FUNCTION_BLOCK MPC_MOVE_BLOCKED_NMPC_V4 (* High-range V4 state-disturbance MPC identified from real 3, 5, 8.5 and 13 cm calibration transients *)
  (* Standard: 61499-2 *)
  (* Version 4.0, 2026-08-29, Guilherme *)
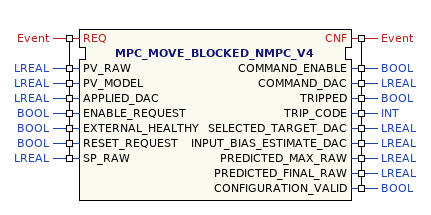
  EVENT_INPUT
    REQ WITH PV_RAW, PV_MODEL, APPLIED_DAC, ENABLE_REQUEST, EXTERNAL_HEALTHY, RESET_REQUEST, SP_RAW; (* Execute one 500 ms high-range MPC V4 cycle *)
  END_EVENT
  EVENT_OUTPUT
    CNF WITH COMMAND_ENABLE, COMMAND_DAC, TRIPPED, TRIP_CODE, SELECTED_TARGET_DAC, INPUT_BIAS_ESTIMATE_DAC, PREDICTED_MAX_RAW, PREDICTED_FINAL_RAW, CONFIGURATION_VALID; (* MPC cycle completed *)
  END_EVENT
  VAR_INPUT
    PV_RAW : LREAL; (* Unfiltered raw level used by the measured hard trip *)
    PV_MODEL : LREAL; (* 9-sample rolling-median raw level used by the identified model *)
    APPLIED_DAC : LREAL; (* PLC-confirmed DAC used as the move-constraint reference *)
    ENABLE_REQUEST : BOOL; (* Explicit operator/commissioning enable; FALSE is normal zero-output mode *)
    EXTERNAL_HEALTHY : BOOL; (* PLC/gateway watchdog healthy input *)
    RESET_REQUEST : BOOL; (* Explicitly clear the latched MPC trip and internal estimator state *)
    SP_RAW : LREAL; (* Raw-count setpoint; 15 cm validation target is 16000 *)
  END_VAR
  VAR_OUTPUT
    COMMAND_ENABLE : BOOL; (* Fail-closed actuator enable request *)
    COMMAND_DAC : LREAL; (* MPC DAC request before downstream defense-in-depth limiting *)
    TRIPPED : BOOL; (* Latched MPC trip state *)
    TRIP_CODE : INT; (* 0=none,1=non-finite input,2=external health,3=PV bounds,4=AppliedDAC bounds,5=setpoint bounds,6=no feasible prediction,7=delay history not ready *)
    SELECTED_TARGET_DAC : LREAL; (* Move-blocked target selected by the current horizon search *)
    INPUT_BIAS_ESTIMATE_DAC : LREAL; (* Bounded offset-compensation estimate *)
    PREDICTED_MAX_RAW : LREAL; (* Maximum predicted model level for the selected candidate *)
    PREDICTED_FINAL_RAW : LREAL; (* Final horizon model level for the selected candidate *)
    CONFIGURATION_VALID : BOOL; (* Frozen V4 high-range configuration is internally valid *)
  END_VAR
  VAR
    trip_latched_internal : BOOL := FALSE;
    trip_code_internal : INT := 0;
    history_count : DINT := 0;
    record_history_internal : BOOL := FALSE;
    best_found : BOOL := FALSE;
    candidate_feasible : BOOL := FALSE;
    h00 : LREAL := 0.0;
    h01 : LREAL := 0.0;
    h02 : LREAL := 0.0;
    h03 : LREAL := 0.0;
    h04 : LREAL := 0.0;
    h05 : LREAL := 0.0;
    h06 : LREAL := 0.0;
    h07 : LREAL := 0.0;
    h08 : LREAL := 0.0;
    h09 : LREAL := 0.0;
    h10 : LREAL := 0.0;
    h11 : LREAL := 0.0;
    h12 : LREAL := 0.0;
    h13 : LREAL := 0.0;
    h14 : LREAL := 0.0;
    h15 : LREAL := 0.0;
    h16 : LREAL := 0.0;
    h17 : LREAL := 0.0;
    q00 : LREAL := 0.0;
    q01 : LREAL := 0.0;
    q02 : LREAL := 0.0;
    q03 : LREAL := 0.0;
    q04 : LREAL := 0.0;
    q05 : LREAL := 0.0;
    q06 : LREAL := 0.0;
    q07 : LREAL := 0.0;
    q08 : LREAL := 0.0;
    q09 : LREAL := 0.0;
    q10 : LREAL := 0.0;
    q11 : LREAL := 0.0;
    q12 : LREAL := 0.0;
    q13 : LREAL := 0.0;
    q14 : LREAL := 0.0;
    q15 : LREAL := 0.0;
    q16 : LREAL := 0.0;
    q17 : LREAL := 0.0;
    best_cost : LREAL := 0.0;
    best_target : LREAL := 0.0;
    best_predicted_max : LREAL := 0.0;
    best_predicted_final : LREAL := 0.0;
    candidate_target : LREAL := 0.0;
    predicted_y : LREAL := 0.0;
    predicted_u : LREAL := 0.0;
    previous_u : LREAL := 0.0;
    delayed_u : LREAL := 0.0;
    candidate_cost : LREAL := 0.0;
    candidate_predicted_max : LREAL := 0.0;
    delta_u : LREAL := 0.0;
    effective_input : LREAL := 0.0;
    phi_value : LREAL := 0.0;
    tracking_error : LREAL := 0.0;
    move_value : LREAL := 0.0;
    soft_excess : LREAL := 0.0;
    terminal_error : LREAL := 0.0;
    command_candidate : LREAL := 0.0;
    candidate_index : DINT := 0;
    prediction_index : DINT := 0;
    disturbance_hat_internal : LREAL := 0.0;
    disturbance_previous_pv_internal : LREAL := 0.0;
    disturbance_previous_valid_internal : BOOL := FALSE;
    disturbance_prediction_internal : LREAL := 0.0;
    disturbance_innovation_internal : LREAL := 0.0;
  END_VAR
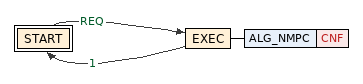
  EC_STATES
    START;
    EXEC : ALG_NMPC -> CNF;
  END_STATES
  EC_TRANSITIONS
    START TO EXEC := REQ;
    EXEC TO START := 1;
  END_TRANSITIONS
  ALGORITHM ALG_NMPC IN ST: (* Move-blocked V4 high-range NMPC with state-disturbance estimation, model constraints, trip latch, and piecewise-linear x^1.2 input *)
IF RESET_REQUEST THEN
    trip_latched_internal := FALSE;
    trip_code_internal := 0;
    disturbance_hat_internal := LREAL#0.0;
    disturbance_previous_pv_internal := LREAL#0.0;
    disturbance_previous_valid_internal := FALSE;
    disturbance_prediction_internal := LREAL#0.0;
    disturbance_innovation_internal := LREAL#0.0;
END_IF;

CONFIGURATION_VALID := TRUE;
COMMAND_ENABLE := FALSE;
COMMAND_DAC := LREAL#0.0;
SELECTED_TARGET_DAC := LREAL#0.0;
INPUT_BIAS_ESTIMATE_DAC := LREAL#0.0;
PREDICTED_MAX_RAW := LREAL#-1.0;
PREDICTED_FINAL_RAW := LREAL#-1.0;

record_history_internal := (PV_RAW = PV_RAW) AND (PV_MODEL = PV_MODEL) AND (APPLIED_DAC = APPLIED_DAC) AND (SP_RAW = SP_RAW) AND (APPLIED_DAC >= LREAL#0.0) AND (APPLIED_DAC <= LREAL#16000.0);

IF NOT trip_latched_internal THEN
    IF NOT ENABLE_REQUEST THEN
        disturbance_hat_internal := LREAL#0.0;
        disturbance_previous_pv_internal := LREAL#0.0;
        disturbance_previous_valid_internal := FALSE;
        disturbance_prediction_internal := LREAL#0.0;
        disturbance_innovation_internal := LREAL#0.0;
        COMMAND_ENABLE := FALSE;
        COMMAND_DAC := LREAL#0.0;
    ELSE
        IF NOT EXTERNAL_HEALTHY THEN
            trip_latched_internal := TRUE;
            trip_code_internal := 2;
        ELSIF NOT (PV_RAW = PV_RAW) OR NOT (PV_MODEL = PV_MODEL) OR NOT (APPLIED_DAC = APPLIED_DAC) OR NOT (SP_RAW = SP_RAW) THEN
            trip_latched_internal := TRUE;
            trip_code_internal := 1;
        ELSIF PV_RAW < LREAL#0.0 OR PV_MODEL < LREAL#0.0 OR PV_RAW >= LREAL#20000.0 THEN
            trip_latched_internal := TRUE;
            trip_code_internal := 3;
        ELSIF APPLIED_DAC < LREAL#0.0 OR APPLIED_DAC > LREAL#16000.0 THEN
            trip_latched_internal := TRUE;
            trip_code_internal := 4;
        ELSIF SP_RAW < LREAL#0.0 OR SP_RAW >= LREAL#18000.0 THEN
            trip_latched_internal := TRUE;
            trip_code_internal := 5;
        ELSE
            IF disturbance_previous_valid_internal THEN
                IF disturbance_previous_pv_internal < LREAL#257.0 THEN
                    disturbance_previous_pv_internal := LREAL#257.0;
                END_IF;
                effective_input := APPLIED_DAC - LREAL#11750.0;
                IF effective_input < LREAL#0.0 THEN
                    effective_input := LREAL#0.0;
                ELSIF effective_input > LREAL#4250.0 THEN
                    effective_input := LREAL#4250.0;
                END_IF;
                IF effective_input <= LREAL#0.0 THEN
                    phi_value := LREAL#0.0;
                ELSIF effective_input <= LREAL#250.0 THEN
                    phi_value := LREAL#0.000000000000000 + LREAL#3.017088168272581 * (effective_input - LREAL#0.0);
                ELSIF effective_input <= LREAL#500.0 THEN
                    phi_value := LREAL#754.272042068145197 + LREAL#3.914360263278881 * (effective_input - LREAL#250.0);
                ELSIF effective_input <= LREAL#750.0 THEN
                    phi_value := LREAL#1732.862107887865477 + LREAL#4.343991804743724 * (effective_input - LREAL#500.0);
                ELSIF effective_input <= LREAL#1000.0 THEN
                    phi_value := LREAL#2818.860059073796492 + LREAL#4.648846585844700 * (effective_input - LREAL#750.0);
                ELSIF effective_input <= LREAL#1250.0 THEN
                    phi_value := LREAL#3981.071705534971443 + LREAL#4.889543362906937 * (effective_input - LREAL#1000.0);
                ELSIF effective_input <= LREAL#1500.0 THEN
                    phi_value := LREAL#5203.457546261705829 + LREAL#5.090329117552494 * (effective_input - LREAL#1250.0);
                ELSIF effective_input <= LREAL#1750.0 THEN
                    phi_value := LREAL#6476.039825649829254 + LREAL#5.263604911708677 * (effective_input - LREAL#1500.0);
                ELSIF effective_input <= LREAL#2000.0 THEN
                    phi_value := LREAL#7791.941053576998456 + LREAL#5.416639939878100 * (effective_input - LREAL#1750.0);
                ELSIF effective_input <= LREAL#2250.0 THEN
                    phi_value := LREAL#9146.101038546523341 + LREAL#5.554090126229741 * (effective_input - LREAL#2000.0);
                ELSIF effective_input <= LREAL#2500.0 THEN
                    phi_value := LREAL#10534.623570103958627 + LREAL#5.679130709085999 * (effective_input - LREAL#2250.0);
                ELSIF effective_input <= LREAL#2750.0 THEN
                    phi_value := LREAL#11954.406247375458406 + LREAL#5.794031214691713 * (effective_input - LREAL#2500.0);
                ELSIF effective_input <= LREAL#3000.0 THEN
                    phi_value := LREAL#13402.914051048386682 + LREAL#5.900474152760405 * (effective_input - LREAL#2750.0);
                ELSIF effective_input <= LREAL#3250.0 THEN
                    phi_value := LREAL#14878.032589238488072 + LREAL#5.999743896709013 * (effective_input - LREAL#3000.0);
                ELSIF effective_input <= LREAL#3500.0 THEN
                    phi_value := LREAL#16377.968563415741301 + LREAL#6.092844710159137 * (effective_input - LREAL#3250.0);
                ELSIF effective_input <= LREAL#3750.0 THEN
                    phi_value := LREAL#17901.179740955525631 + LREAL#6.180577736426479 * (effective_input - LREAL#3500.0);
                ELSIF effective_input <= LREAL#4000.0 THEN
                    phi_value := LREAL#19446.324175062145514 + LREAL#6.263593040671942 * (effective_input - LREAL#3750.0);
                ELSIF effective_input <= LREAL#4250.0 THEN
                    phi_value := LREAL#21012.222435230130941 + LREAL#6.342425861622032 * (effective_input - LREAL#4000.0);
                ELSE
                    phi_value := LREAL#22597.828900635639002;
                END_IF;
                disturbance_prediction_internal := LREAL#257.0 + LREAL#0.997231776304349 * (disturbance_previous_pv_internal - LREAL#257.0) + LREAL#0.004607840412330 * phi_value;
                disturbance_innovation_internal := PV_MODEL - disturbance_prediction_internal;
                disturbance_hat_internal := LREAL#0.9 * disturbance_hat_internal + LREAL#0.1 * disturbance_innovation_internal;
                IF disturbance_hat_internal > LREAL#10.0 THEN
                    disturbance_hat_internal := LREAL#10.0;
                ELSIF disturbance_hat_internal < LREAL#-10.0 THEN
                    disturbance_hat_internal := LREAL#-10.0;
                END_IF;
            END_IF;
            disturbance_previous_pv_internal := PV_MODEL;
            disturbance_previous_valid_internal := TRUE;
            best_found := FALSE;
            best_cost := LREAL#1000000000.0;
            best_target := LREAL#0.0;
            best_predicted_max := LREAL#-1.0;
            best_predicted_final := LREAL#-1.0;
            FOR candidate_index := 0 TO 10 DO
                CASE candidate_index OF
                    0:
                        candidate_target := LREAL#0.0;
                    1:
                        candidate_target := LREAL#12000.0;
                    2:
                        candidate_target := LREAL#12500.0;
                    3:
                        candidate_target := LREAL#13000.0;
                    4:
                        candidate_target := LREAL#13500.0;
                    5:
                        candidate_target := LREAL#13800.0;
                    6:
                        candidate_target := LREAL#14000.0;
                    7:
                        candidate_target := LREAL#14500.0;
                    8:
                        candidate_target := LREAL#15000.0;
                    9:
                        candidate_target := LREAL#15500.0;
                    10:
                        candidate_target := LREAL#16000.0;
                    ELSE
                        candidate_target := LREAL#0.0;
                END_CASE;
                q00 := h00;
                q01 := h01;
                q02 := h02;
                q03 := h03;
                q04 := h04;
                q05 := h05;
                q06 := h06;
                q07 := h07;
                q08 := h08;
                q09 := h09;
                q10 := h10;
                q11 := h11;
                q12 := h12;
                q13 := h13;
                q14 := h14;
                q15 := h15;
                q16 := h16;
                q17 := h17;
                IF PV_MODEL < LREAL#257.0 THEN
                    predicted_y := LREAL#257.0;
                ELSE
                    predicted_y := PV_MODEL;
                END_IF;
                predicted_u := APPLIED_DAC;
                previous_u := APPLIED_DAC;
                candidate_cost := LREAL#0.0;
                candidate_predicted_max := predicted_y;
                candidate_feasible := TRUE;
                FOR prediction_index := 1 TO 60 DO
                    IF candidate_feasible THEN
                        delta_u := candidate_target - predicted_u;
                        IF delta_u > LREAL#750.0 THEN
                            delta_u := LREAL#750.0;
                        ELSIF delta_u < LREAL#-750.0 THEN
                            delta_u := LREAL#-750.0;
                        END_IF;
                        predicted_u := predicted_u + delta_u;
                        IF predicted_u > LREAL#16000.0 THEN
                            predicted_u := LREAL#16000.0;
                        ELSIF predicted_u < LREAL#0.0 THEN
                            predicted_u := LREAL#0.0;
                        END_IF;
                        delayed_u := predicted_u;
                        q00 := q01;
                        q01 := q02;
                        q02 := q03;
                        q03 := q04;
                        q04 := q05;
                        q05 := q06;
                        q06 := q07;
                        q07 := q08;
                        q08 := q09;
                        q09 := q10;
                        q10 := q11;
                        q11 := q12;
                        q12 := q13;
                        q13 := q14;
                        q14 := q15;
                        q15 := q16;
                        q16 := q17;
                        q17 := predicted_u;
                        effective_input := delayed_u - LREAL#11750.0;
                        IF effective_input < LREAL#0.0 THEN
                            effective_input := LREAL#0.0;
                        ELSIF effective_input > LREAL#4250.0 THEN
                            effective_input := LREAL#4250.0;
                        END_IF;
                        IF effective_input <= LREAL#0.0 THEN
                            phi_value := LREAL#0.0;
                        ELSIF effective_input <= LREAL#250.0 THEN
                            phi_value := LREAL#0.000000000000000 + LREAL#3.017088168272581 * (effective_input - LREAL#0.0);
                        ELSIF effective_input <= LREAL#500.0 THEN
                            phi_value := LREAL#754.272042068145197 + LREAL#3.914360263278881 * (effective_input - LREAL#250.0);
                        ELSIF effective_input <= LREAL#750.0 THEN
                            phi_value := LREAL#1732.862107887865477 + LREAL#4.343991804743724 * (effective_input - LREAL#500.0);
                        ELSIF effective_input <= LREAL#1000.0 THEN
                            phi_value := LREAL#2818.860059073796492 + LREAL#4.648846585844700 * (effective_input - LREAL#750.0);
                        ELSIF effective_input <= LREAL#1250.0 THEN
                            phi_value := LREAL#3981.071705534971443 + LREAL#4.889543362906937 * (effective_input - LREAL#1000.0);
                        ELSIF effective_input <= LREAL#1500.0 THEN
                            phi_value := LREAL#5203.457546261705829 + LREAL#5.090329117552494 * (effective_input - LREAL#1250.0);
                        ELSIF effective_input <= LREAL#1750.0 THEN
                            phi_value := LREAL#6476.039825649829254 + LREAL#5.263604911708677 * (effective_input - LREAL#1500.0);
                        ELSIF effective_input <= LREAL#2000.0 THEN
                            phi_value := LREAL#7791.941053576998456 + LREAL#5.416639939878100 * (effective_input - LREAL#1750.0);
                        ELSIF effective_input <= LREAL#2250.0 THEN
                            phi_value := LREAL#9146.101038546523341 + LREAL#5.554090126229741 * (effective_input - LREAL#2000.0);
                        ELSIF effective_input <= LREAL#2500.0 THEN
                            phi_value := LREAL#10534.623570103958627 + LREAL#5.679130709085999 * (effective_input - LREAL#2250.0);
                        ELSIF effective_input <= LREAL#2750.0 THEN
                            phi_value := LREAL#11954.406247375458406 + LREAL#5.794031214691713 * (effective_input - LREAL#2500.0);
                        ELSIF effective_input <= LREAL#3000.0 THEN
                            phi_value := LREAL#13402.914051048386682 + LREAL#5.900474152760405 * (effective_input - LREAL#2750.0);
                        ELSIF effective_input <= LREAL#3250.0 THEN
                            phi_value := LREAL#14878.032589238488072 + LREAL#5.999743896709013 * (effective_input - LREAL#3000.0);
                        ELSIF effective_input <= LREAL#3500.0 THEN
                            phi_value := LREAL#16377.968563415741301 + LREAL#6.092844710159137 * (effective_input - LREAL#3250.0);
                        ELSIF effective_input <= LREAL#3750.0 THEN
                            phi_value := LREAL#17901.179740955525631 + LREAL#6.180577736426479 * (effective_input - LREAL#3500.0);
                        ELSIF effective_input <= LREAL#4000.0 THEN
                            phi_value := LREAL#19446.324175062145514 + LREAL#6.263593040671942 * (effective_input - LREAL#3750.0);
                        ELSIF effective_input <= LREAL#4250.0 THEN
                            phi_value := LREAL#21012.222435230130941 + LREAL#6.342425861622032 * (effective_input - LREAL#4000.0);
                        ELSE
                            phi_value := LREAL#22597.828900635639002;
                        END_IF;
                        predicted_y := LREAL#257.0 + LREAL#0.997231776304349 * (predicted_y - LREAL#257.0) + LREAL#0.004607840412330 * phi_value + disturbance_hat_internal;
                        IF predicted_y > candidate_predicted_max THEN
                            candidate_predicted_max := predicted_y;
                        END_IF;
                        IF NOT (predicted_y = predicted_y) OR predicted_y > LREAL#19500.0 THEN
                            candidate_feasible := FALSE;
                        ELSE
                            tracking_error := predicted_y - SP_RAW;
                            move_value := predicted_u - previous_u;
                            candidate_cost := candidate_cost + LREAL#5.0 * tracking_error * tracking_error + LREAL#0.00004 * move_value * move_value;
                            IF predicted_y > LREAL#18000.0 THEN
                                soft_excess := predicted_y - LREAL#18000.0;
                                candidate_cost := candidate_cost + LREAL#100.0 * soft_excess * soft_excess;
                            END_IF;
                            previous_u := predicted_u;
                        END_IF;
                    END_IF;
                END_FOR;
                IF candidate_feasible THEN
                    terminal_error := predicted_y - SP_RAW;
                    candidate_cost := candidate_cost + LREAL#10.0 * terminal_error * terminal_error;
                    IF (NOT best_found) OR candidate_cost < best_cost THEN
                        best_found := TRUE;
                        best_cost := candidate_cost;
                        best_target := candidate_target;
                        best_predicted_max := candidate_predicted_max;
                        best_predicted_final := predicted_y;
                    END_IF;
                END_IF;
            END_FOR;
            IF NOT best_found THEN
                trip_latched_internal := TRUE;
                trip_code_internal := 6;
            ELSE
                delta_u := best_target - APPLIED_DAC;
                IF delta_u > LREAL#750.0 THEN
                    delta_u := LREAL#750.0;
                ELSIF delta_u < LREAL#-750.0 THEN
                    delta_u := LREAL#-750.0;
                END_IF;
                command_candidate := APPLIED_DAC + delta_u;
                IF command_candidate > LREAL#16000.0 THEN
                    command_candidate := LREAL#16000.0;
                ELSIF command_candidate < LREAL#0.0 THEN
                    command_candidate := LREAL#0.0;
                END_IF;
                COMMAND_ENABLE := TRUE;
                COMMAND_DAC := command_candidate;
                SELECTED_TARGET_DAC := best_target;
                PREDICTED_MAX_RAW := best_predicted_max;
                PREDICTED_FINAL_RAW := best_predicted_final;
            END_IF;
        END_IF;
    END_IF;
END_IF;

IF record_history_internal THEN
    h00 := h01;
    h01 := h02;
    h02 := h03;
    h03 := h04;
    h04 := h05;
    h05 := h06;
    h06 := h07;
    h07 := h08;
    h08 := h09;
    h09 := h10;
    h10 := h11;
    h11 := h12;
    h12 := h13;
    h13 := h14;
    h14 := h15;
    h15 := h16;
    h16 := h17;
    h17 := APPLIED_DAC;
    IF history_count < 18 THEN
        history_count := history_count + 1;
    END_IF;
END_IF;

TRIPPED := trip_latched_internal;
TRIP_CODE := trip_code_internal;
INPUT_BIAS_ESTIMATE_DAC := LREAL#0.0;

IF trip_latched_internal THEN
    COMMAND_ENABLE := FALSE;
    COMMAND_DAC := LREAL#0.0;
    SELECTED_TARGET_DAC := LREAL#0.0;
    PREDICTED_MAX_RAW := LREAL#-1.0;
    PREDICTED_FINAL_RAW := LREAL#-1.0;
END_IF;
  END_ALGORITHM
END_FUNCTION_BLOCK
